FUNCTION_BLOCK manutencao (* Basic Function Block Type *)
  (* Standard: 61499-2 *)
  (* Version 0.0, 26/02/2026, Template *)
  PACKAGE Hidryco.HidrycoLib;
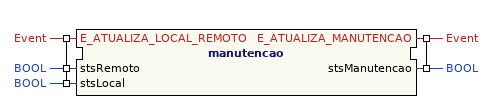
  EVENT_INPUT
    E_ATUALIZA_LOCAL_REMOTO WITH stsRemoto, stsLocal;
  END_EVENT
  EVENT_OUTPUT
    E_ATUALIZA_MANUTENCAO WITH stsManutencao;
  END_EVENT
  VAR_INPUT
    stsRemoto : BOOL;
    stsLocal : BOOL;
  END_VAR
  VAR_OUTPUT
    stsManutencao : BOOL;
  END_VAR
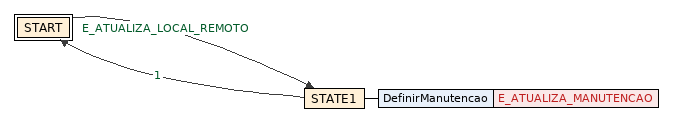
  EC_STATES
    START; (* Initial State *)
    STATE1 : DefinirManutencao -> E_ATUALIZA_MANUTENCAO;
  END_STATES
  EC_TRANSITIONS
    START TO STATE1 := E_ATUALIZA_LOCAL_REMOTO;
    STATE1 TO START := 1;
  END_TRANSITIONS
  ALGORITHM DefinirManutencao IN ST:
IF NOT stsLocal AND NOT stsRemoto THEN
	stsManutencao := TRUE;
ELSE
	stsManutencao := FALSE;
END_IF;
;
  END_ALGORITHM
END_FUNCTION_BLOCK
